{attribute 'linkalways'}
{attribute 'hide_all_locals'}
FUNCTION_BLOCK ValueTod EXTENDS ValueTodRead IMPLEMENTS Value
VAR
END_VAR

METHOD SetFromType : BOOL
VAR_INPUT
	source : __SYSTEM.AnyType;
END_VAR
SetFromType := ConvertAnyType(source, thisAnyType);
END_METHOD

METHOD SetFromString : BOOL
VAR_INPUT
	value : T_MaxString;
END_VAR
thisValue := STRING_TO_TOD(value);

SetFromString := TRUE;
END_METHOD

METHOD Set : BOOL
VAR_INPUT
	source : ANY;
END_VAR
Set := ConvertAnyType(source, thisAnyType);
END_METHOD

END_FUNCTION_BLOCK

(* stored: Version 1.1.0.1
   POU ValueTod: Id {192476c2-d0a4-417e-af0a-5f2e79c272a3}, SpecialFunc None
   Method SetFromType: Id {5da1e449-6dcb-45e5-8687-c3f67f61f777}
   Method SetFromString: Id {bf98508c-8fee-4c2f-b80a-1a2122ab4b6d}
   Method Set: Id {d297a4e3-88cb-4105-b069-680f272f66d2} *)
